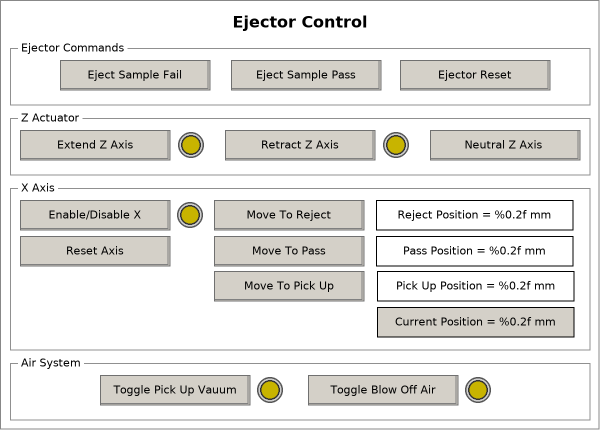
VISUALIZATION Manual_Ejector  // 600x430
    GroupBox (10,355 580x65), "Air System"
    Label (0,7 600x30), "Ejector Control"
    Button (100,375 150x30), "Toggle Pick Up Vauum"
        OnMouseClick: execute { MAIN.fbSlitter.Manual.bEjectVacuum := TRUE; }
    Button (308,375 150x30), "Toggle Blow Off Air"
        OnMouseClick: execute { MAIN.fbSlitter.Manual.bEjectBlowOff := TRUE; }
    Lamp1 (463,375 30x30), variable: MAIN.fbSlitter.Ejector._BlowOff, style: Lamp-Lamp1-Yellow
    Lamp1 (255,375 30x30), variable: MAIN.fbSlitter.Ejector._Vacuum, style: Lamp-Lamp1-Yellow
    Group (10,110 580x65)
        GroupBox (0,0 580x65), "Z Actuator"
        Button (10,20 150x30), "Extend Z Axis", input disabled if: MAIN.fbSlitter.bBusy
            OnMouseClick: execute { MAIN.fbSlitter.Manual.bEjectZExtend := TRUE; }
        Button (215,20 150x30), "Retract Z Axis", input disabled if: MAIN.fbSlitter.bBusy
            OnMouseClick: execute { MAIN.fbSlitter.Manual.bEjectZRetract := TRUE; }
        Button (420,20 150x30), "Neutral Z Axis", input disabled if: MAIN.fbSlitter.bBusy
            tap MAIN.fbSlitter.Manual.bEjectZOff
            OnMouseClick: execute { MAIN.fbSlitter.Manual.bEjectZNeutral := TRUE; }
        Lamp1 (166,20 30x30), variable: MAIN.fbSlitter.Ejector.zSlide.diExtended, style: Lamp-Lamp1-Yellow
        Lamp1 (371,20 30x30), variable: MAIN.fbSlitter.Ejector.zSlide.diRetracted, style: Lamp-Lamp1-Yellow
    GroupBox (10,40 580x65), "Ejector Commands"
        Button (390,20 150x30), "Ejector Reset", input disabled if: MAIN.fbSlitter.bBusy
            OnMouseClick: execute { MAIN.fbSlitter.Manual.bEjectReset := TRUE; }
    Button (60,60 150x30), "Eject Sample Fail", input disabled if: MAIN.fbSlitter.bBusy
        OnMouseClick: execute { MAIN.fbSlitter.Manual.bEjectSampleFail := TRUE; }
    Button (231,60 150x30), "Eject Sample Pass", input disabled if: MAIN.fbSlitter.bBusy
        OnMouseClick: execute { MAIN.fbSlitter.Manual.bEjectSamplePass := TRUE; }
    GroupBox (10,180 580x170), "X Axis"
        Rectangle (367,91 197x30), "Pick Up Position = %0.2f mm", text variable: MAIN.fbSlitter.Ejector._hmiParameters.ejectPositionHome
            OnMouseClick: write MAIN.fbSlitter.Ejector._hmiParameters.ejectPositionHome via Default, title 'Pick Up Position'
        Rectangle (367,127 197x30), "Current Position = %0.2f mm", text variable: MAIN.fbSlitter.Ejector.axis.axis.NcToPlc.ActPos
        Button (10,56 150x30), "Reset Axis"
            OnMouseClick: execute { MAIN.fbSlitter.Manual.bEjectAxisReset := TRUE; }
    Button (20,200 150x30), "Enable/Disable X", input disabled if: MAIN.fbSlitter.bBusy
        OnMouseClick: execute { MAIN.fbSlitter.Manual.bEjectAxisEnableToggle := TRUE; }
    Lamp1 (175,200 30x30), variable: MAIN.fbSlitter.Ejector.axis.axis.NcToPlc.StateDWord.0 = 1, style: Lamp-Lamp1-Yellow
    Button (214,200 150x30), "Move To Reject", input disabled if: MAIN.fbSlitter.bBusy
        OnMouseClick: execute { Main.fbSlitter.Manual.bEjectAxisFailPosition := TRUE; }
    Button (214,236 150x30), "Move To Pass", input disabled if: MAIN.fbSlitter.bBusy
        OnMouseClick: execute { Main.fbSlitter.Manual.bEjectAxisPassPosition := TRUE; }
    Button (214,271 150x30), "Move To Pick Up", input disabled if: MAIN.fbSlitter.bBusy
        OnMouseClick: execute { Main.fbSlitter.Manual.bEjectAxisHomePosition := TRUE; }
    Rectangle (376,200 197x30), "Reject Position = %0.2f mm", text variable: MAIN.fbSlitter.Ejector._hmiParameters.ejectPositionFail
        OnMouseClick: write MAIN.fbSlitter.Ejector._hmiParameters.ejectPositionFail via Default, title 'Reject Position'
    Rectangle (376,236 197x30), "Pass Position = %0.2f mm", text variable: MAIN.fbSlitter.Ejector._hmiParameters.ejectPositionPass
        OnMouseClick: write MAIN.fbSlitter.Ejector._hmiParameters.ejectPositionPass via Default, title 'Pass Position'
END_VISUALIZATION

(* stored: Version 1.1.0.1, ProductVersion 3.1.4024.9
   Visu Manual_Ejector: Id {eddb5234-c01d-4932-a26b-704fb44aae16} *)
